# EPICS substitutions: WS3122App/Db/ws3122.substitutions
file WS3122Base.template {
pattern { P, R, PORT }
{ "$(P)", "$(R)", "$(PORT)"}
}

file BasicWave.template {
pattern { P, R, PORT }
{ "$(P)", "$(R)", "$(PORT)"}
}
